TYPE
    ST_Indicator_Config : STRUCT
        PulseOnTime  : LREAL;
        PulseOffTime : LREAL;
    END_STRUCT
END_TYPE

(* stored: Version 1.1.0.1
   DUT ST_Indicator_Config: Id {a19a0e99-e216-4ff3-836f-dd13d4549e9d} *)
